Staubli VAL3: start.pgx

program start()
begin

  //测试开始
  call moveTest()


end
